(* Logix 5000 project; controller NSH_PLC1 vendor 1 type 14 code 167 rev 32.11; software revision 32.02; part 2 of 12 *)
(* tags used below, declared in another part *)
   FaultReset : BOOL;   // Huller-Sheller Fault Reset
   Num_Faults : DINT;   // Number of Huller-Sheller Faults
   Num_Warnings : DINT;   // Number of Huller-Sheller Warnings
   TempCommAlarm : BOOL;   // Temp Motor, AOP communications Alarm
   TempImbalanceTrip : BOOL;   // Temp Motor, Phase Imbalance Trip
   TempImbalanceWarning : BOOL;   // Temp Motor, Phase Imbalance Warning
   TempMotor : Motor;   // Temp Motor Tag for Subroutines
   TempOverloadTrip : BOOL;   // Temp Motor, Overload Trip
   TempOverloadWarning : BOOL;   // Temp Motor, Overlaod Warning
   TempPhaseLossTrip : BOOL;   // Temp Motor, Phase Loss Trip
   TempReady : BOOL;   // Temp Motor is ready
   TempRunning : BOOL;   // Temp Motor is Running
   TempTriped : BOOL;   // Temp Motor Tripped
   TempWarning : BOOL;   // Temp Motor Warning
   AFI : BOOL;   // Always False
   BH1 : Motor;   // Auger
   BH1D : Motor;   // Airlock
   BH2 : Motor;   // S. Ele
   BH2D : Motor;   // Airlock
   BH3D : Motor;   // Airlock
   C10 : Motor;   // Auger
   C1A : Motor;   // Auger
   C1B : Motor;   // Auger
   C2 : Motor;   // Auger
   C3A : Motor;   // Auger
   C3B : Motor;   // Auger
   C4 : Motor;   // Ele.
   C7 : Motor;   // Ele
   C8 : Motor;   // Auger
   C9 : Motor;   // Auger
   CL1 : Motor;   // Auger
   CL2 : Motor;   // Auger
   CL3 : Motor;   // Auger
   CL4 : Motor;   // Auger
   CL5 : Motor;   // Auger
   CL6 : Motor;   // Auger
   D10 : Motor;   // Ele
   D11 : Motor;   // Auger
   D12 : Motor;   // Auger
   D13 : Motor;   // Auger
   D14 : Motor;   // Auger
   D1A : Motor;   // Auger
   D1B : Motor;   // Auger
   D2 : Motor;   // Auger
   D4 : Motor;   // Auger
   D5 : Motor;   // Auger
   D6 : Motor;   // Auger
   DL1 : Motor;   // Auger
   M20 : Motor;   // Ele.
   M21 : Motor;   // Nolin
   M25 : Motor;   // Accept Vib.
   M42C : Motor;   // 3C Deck
   M42D : Motor;   // 3C Deck
   M43CA : Motor;   // Asp.
   M43CB : Motor;   // Asp.
   M43DA : Motor;   // Asp.
   M43DB : Motor;   // Asp.
   S11 : Motor;   // Ele.
   S12 : Motor;   // Auger
   S47 : Motor;   // Auger
   S48 : Motor;   // Auger
   S49 : Motor;   // Auger
   S50 : Motor;   // Auger
   SL1 : Motor;   // Auger
   T1 : Motor;   // Belt
   T2 : Motor;   // Belt
   T3 : Motor;   // Belt
   TMR_StartHS : TIMER;   // Run Hullers & Shellers Warning Timer
(* HullerSheller, continued *)

ROUTINE E300_StatusAlmWarnSUB   (* ladder *)
// Decode Status Bits and Set Warnings and Alarms For NRFV Motors with E300
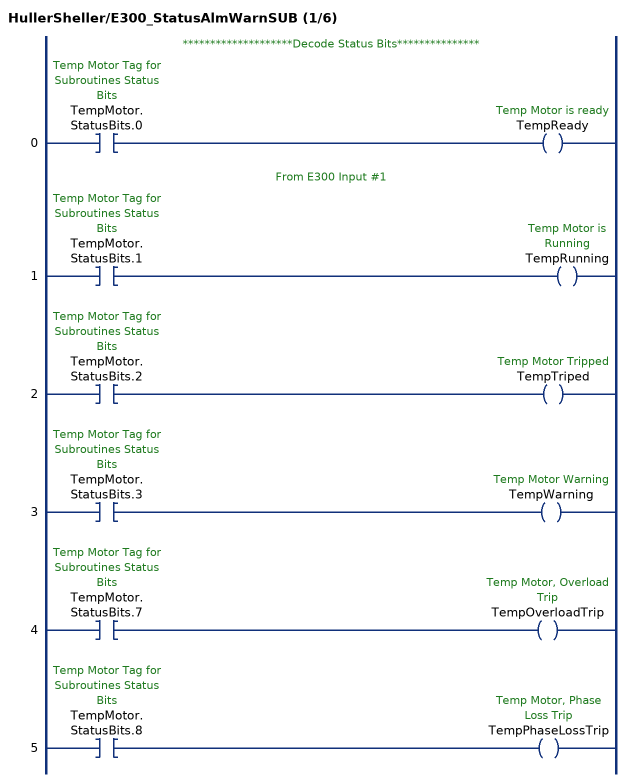
   // ********************Decode Status Bits***************
   0: XIC(TempMotor.StatusBits.0)OTE(TempReady);
   // From E300 Input #1
   1: XIC(TempMotor.StatusBits.1)OTE(TempRunning);
   2: XIC(TempMotor.StatusBits.2)OTE(TempTriped);
   3: XIC(TempMotor.StatusBits.3)OTE(TempWarning);
   4: XIC(TempMotor.StatusBits.7)OTE(TempOverloadTrip);
   5: XIC(TempMotor.StatusBits.8)OTE(TempPhaseLossTrip);
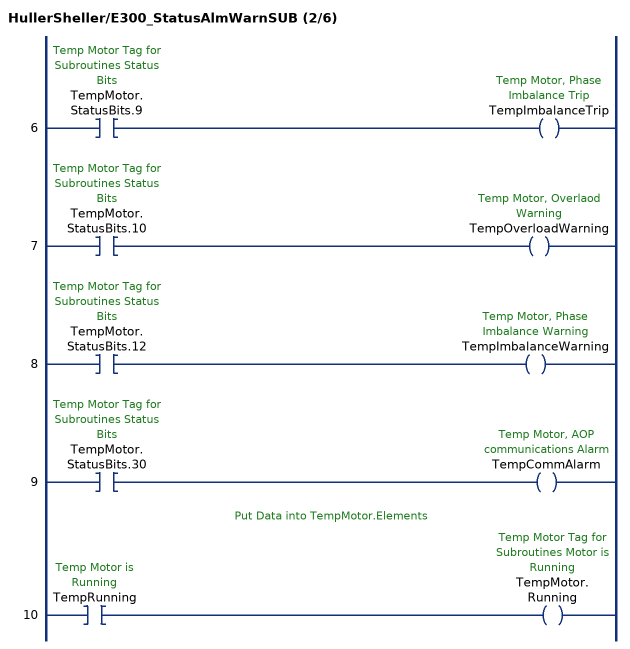
   6: XIC(TempMotor.StatusBits.9)OTE(TempImbalanceTrip);
   7: XIC(TempMotor.StatusBits.10)OTE(TempOverloadWarning);
   8: XIC(TempMotor.StatusBits.12)OTE(TempImbalanceWarning);
   9: XIC(TempMotor.StatusBits.30)OTE(TempCommAlarm);
   // Put Data into TempMotor.Elements
   10: XIC(TempRunning)OTE(TempMotor.Running);
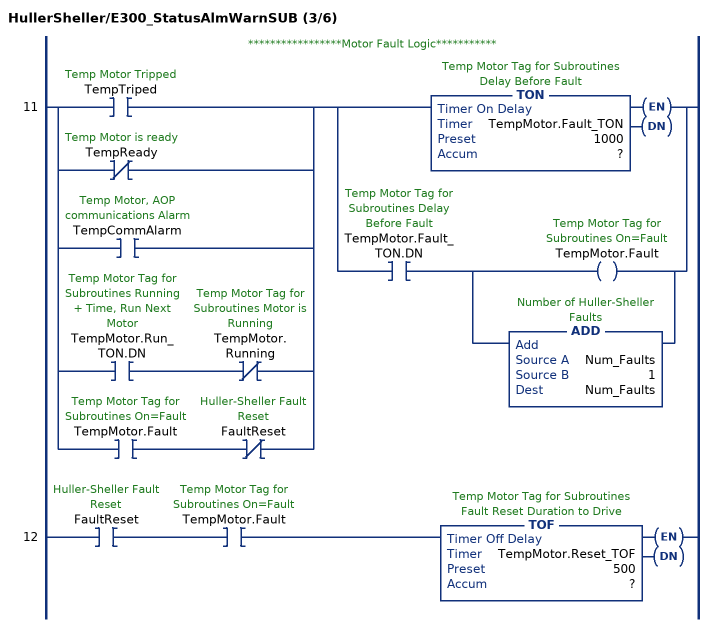
   // *****************Motor Fault Logic***********
   11: [XIC(TempTriped) ,XIO(TempReady) ,XIC(TempCommAlarm) ,XIC(TempMotor.Run_TON.DN) XIO(TempMotor.Running) ,XIC(TempMotor.Fault) XIO(FaultReset) ][TON(TempMotor.Fault_TON,?,?) ,XIC(TempMotor.Fault_TON.DN) [OTE(TempMotor.Fault) ,ADD(Num_Faults,1,Num_Faults) ] ];
   12: XIC(FaultReset)XIC(TempMotor.Fault)TOF(TempMotor.Reset_TOF,?,?);
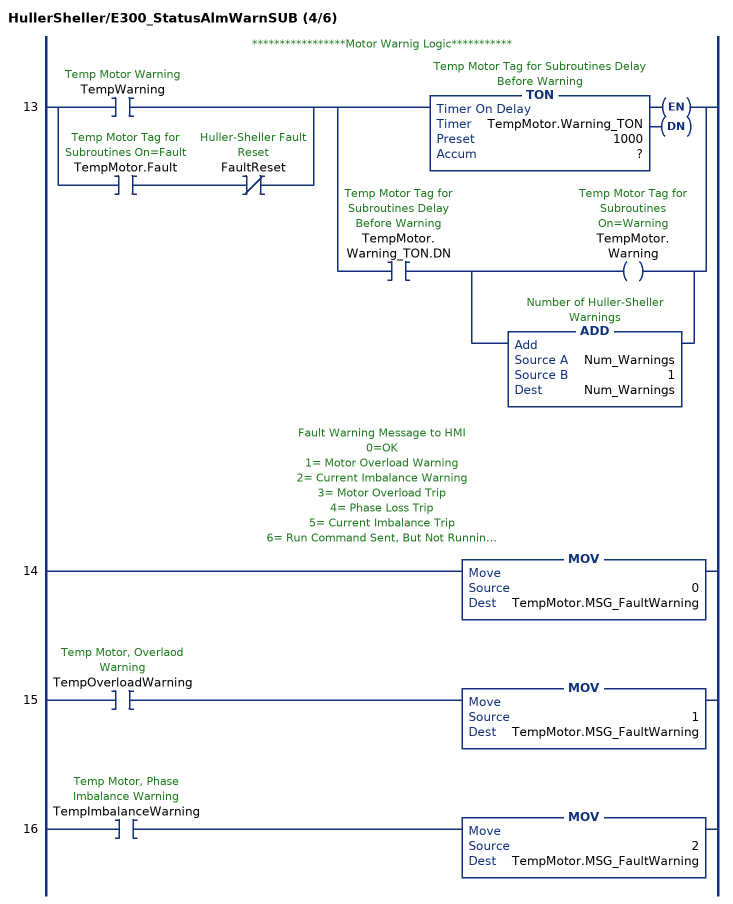
   // *****************Motor Warnig Logic***********
   13: [XIC(TempWarning) ,XIC(TempMotor.Fault) XIO(FaultReset) ][TON(TempMotor.Warning_TON,?,?) ,XIC(TempMotor.Warning_TON.DN) [OTE(TempMotor.Warning) ,ADD(Num_Warnings,1,Num_Warnings) ] ];
   // Fault Warning Message to HMI
   // 0=OK
   // 1= Motor Overload Warning
   // 2= Current Imbalance Warning
   // 3= Motor Overload Trip
   // 4= Phase Loss Trip
   // 5= Current Imbalance Trip
   // 6= Run Command Sent, But Not Running
   // 7=Loss Of Ethernet Communications
   // 8=VFD Fault
   14: MOV(0,TempMotor.MSG_FaultWarning);
   15: XIC(TempOverloadWarning)MOV(1,TempMotor.MSG_FaultWarning);
   16: XIC(TempImbalanceWarning)MOV(2,TempMotor.MSG_FaultWarning);
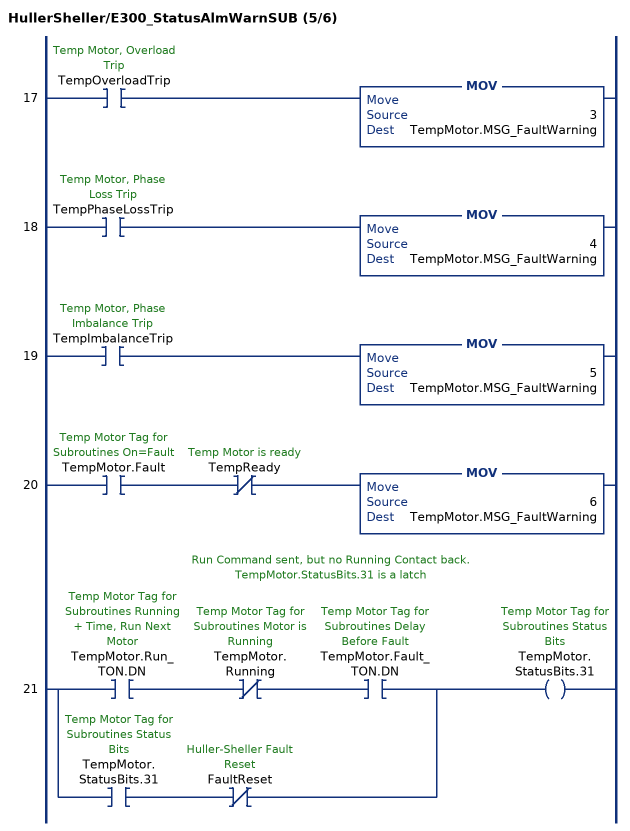
   17: XIC(TempOverloadTrip)MOV(3,TempMotor.MSG_FaultWarning);
   18: XIC(TempPhaseLossTrip)MOV(4,TempMotor.MSG_FaultWarning);
   19: XIC(TempImbalanceTrip)MOV(5,TempMotor.MSG_FaultWarning);
   20: XIC(TempMotor.Fault)XIO(TempReady)MOV(6,TempMotor.MSG_FaultWarning);
   // Run Command sent, but no Running Contact back.
   // TempMotor.StatusBits.31 is a latch
   21: [XIC(TempMotor.Run_TON.DN) XIO(TempMotor.Running) XIC(TempMotor.Fault_TON.DN) ,XIC(TempMotor.StatusBits.31) XIO(FaultReset) ]OTE(TempMotor.StatusBits.31);
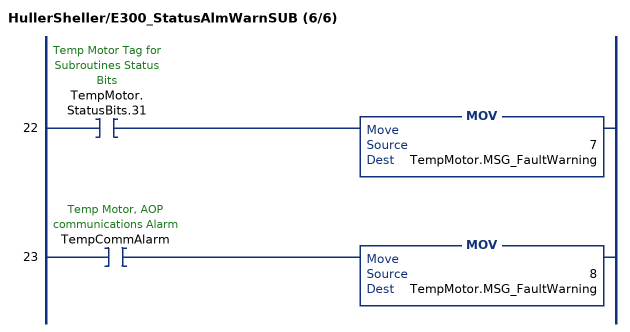
   22: XIC(TempMotor.StatusBits.31)MOV(7,TempMotor.MSG_FaultWarning);
   23: XIC(TempCommAlarm)MOV(8,TempMotor.MSG_FaultWarning);
END_ROUTINE

ROUTINE HS_MainJSR   (* ladder *)
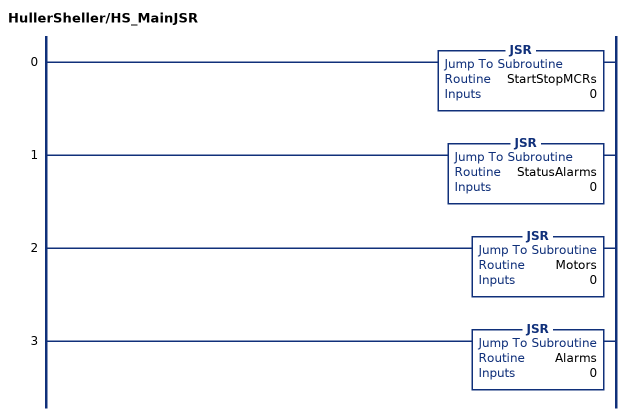
   0: JSR(StartStopMCRs,0);
   1: JSR(StatusAlarms,0);
   2: JSR(Motors,0);
   3: JSR(Alarms,0);
END_ROUTINE

ROUTINE Motors   (* ladder *)
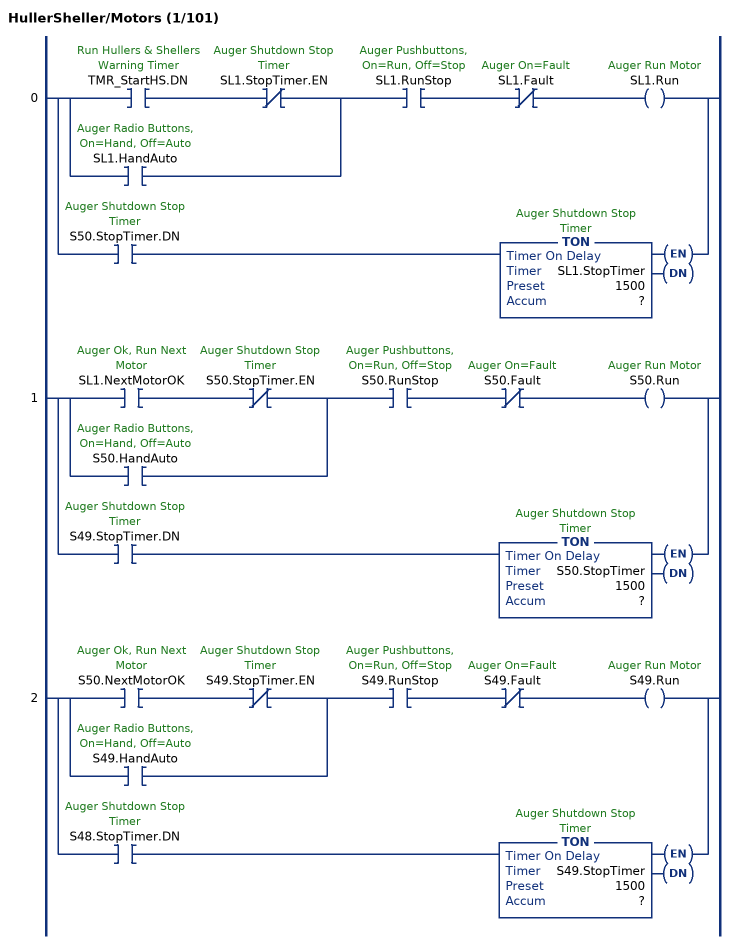
   0: [[XIC(TMR_StartHS.DN) XIO(SL1.StopTimer.EN) ,XIC(SL1.HandAuto) ] XIC(SL1.RunStop) XIO(SL1.Fault) OTE(SL1.Run) ,XIC(S50.StopTimer.DN) TON(SL1.StopTimer,?,?) ];
   1: [[XIC(SL1.NextMotorOK) XIO(S50.StopTimer.EN) ,XIC(S50.HandAuto) ] XIC(S50.RunStop) XIO(S50.Fault) OTE(S50.Run) ,XIC(S49.StopTimer.DN) TON(S50.StopTimer,?,?) ];
   2: [[XIC(S50.NextMotorOK) XIO(S49.StopTimer.EN) ,XIC(S49.HandAuto) ] XIC(S49.RunStop) XIO(S49.Fault) OTE(S49.Run) ,XIC(S48.StopTimer.DN) TON(S49.StopTimer,?,?) ];
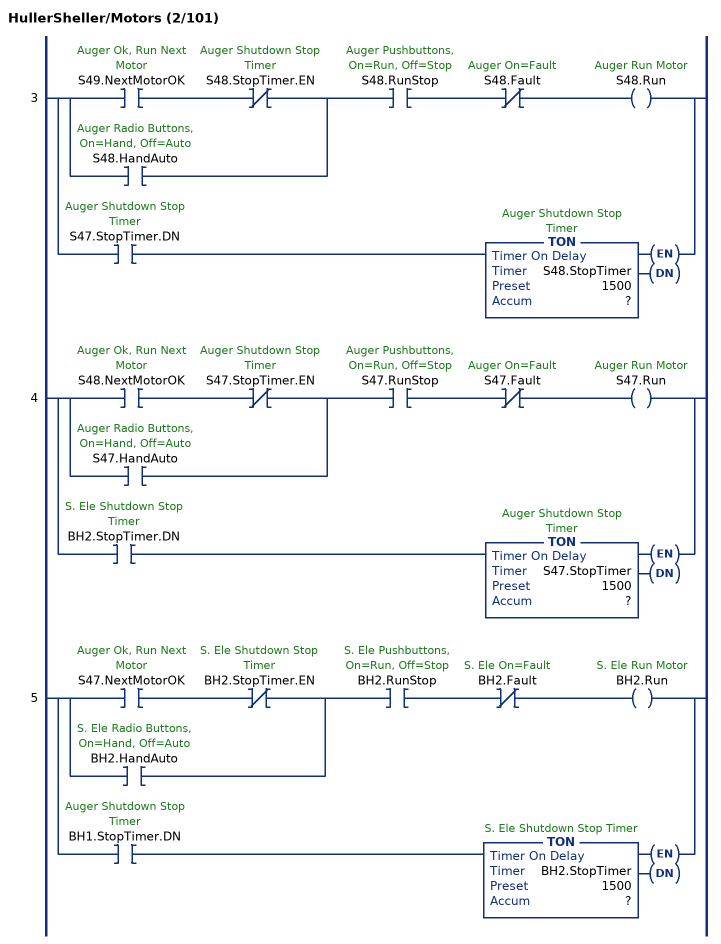
   3: [[XIC(S49.NextMotorOK) XIO(S48.StopTimer.EN) ,XIC(S48.HandAuto) ] XIC(S48.RunStop) XIO(S48.Fault) OTE(S48.Run) ,XIC(S47.StopTimer.DN) TON(S48.StopTimer,?,?) ];
   4: [[XIC(S48.NextMotorOK) XIO(S47.StopTimer.EN) ,XIC(S47.HandAuto) ] XIC(S47.RunStop) XIO(S47.Fault) OTE(S47.Run) ,XIC(BH2.StopTimer.DN) TON(S47.StopTimer,?,?) ];
   5: [[XIC(S47.NextMotorOK) XIO(BH2.StopTimer.EN) ,XIC(BH2.HandAuto) ] XIC(BH2.RunStop) XIO(BH2.Fault) OTE(BH2.Run) ,XIC(BH1.StopTimer.DN) TON(BH2.StopTimer,?,?) ];
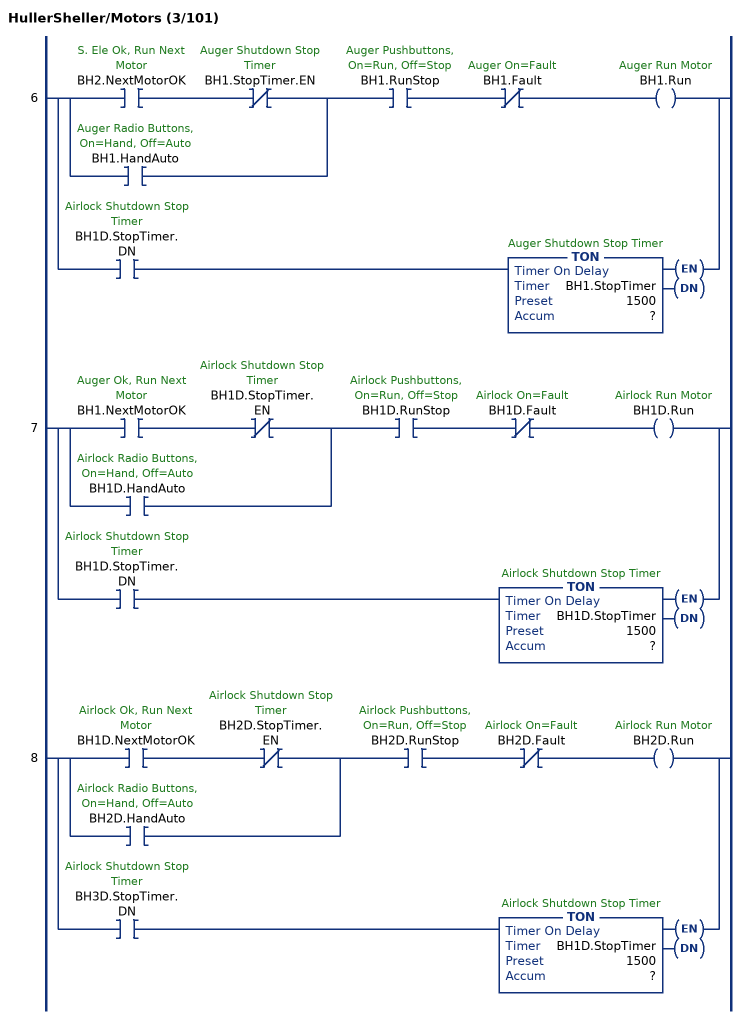
   6: [[XIC(BH2.NextMotorOK) XIO(BH1.StopTimer.EN) ,XIC(BH1.HandAuto) ] XIC(BH1.RunStop) XIO(BH1.Fault) OTE(BH1.Run) ,XIC(BH1D.StopTimer.DN) TON(BH1.StopTimer,?,?) ];
   7: [[XIC(BH1.NextMotorOK) XIO(BH1D.StopTimer.EN) ,XIC(BH1D.HandAuto) ] XIC(BH1D.RunStop) XIO(BH1D.Fault) OTE(BH1D.Run) ,XIC(BH1D.StopTimer.DN) TON(BH1D.StopTimer,?,?) ];
   8: [[XIC(BH1D.NextMotorOK) XIO(BH2D.StopTimer.EN) ,XIC(BH2D.HandAuto) ] XIC(BH2D.RunStop) XIO(BH2D.Fault) OTE(BH2D.Run) ,XIC(BH3D.StopTimer.DN) TON(BH1D.StopTimer,?,?) ];
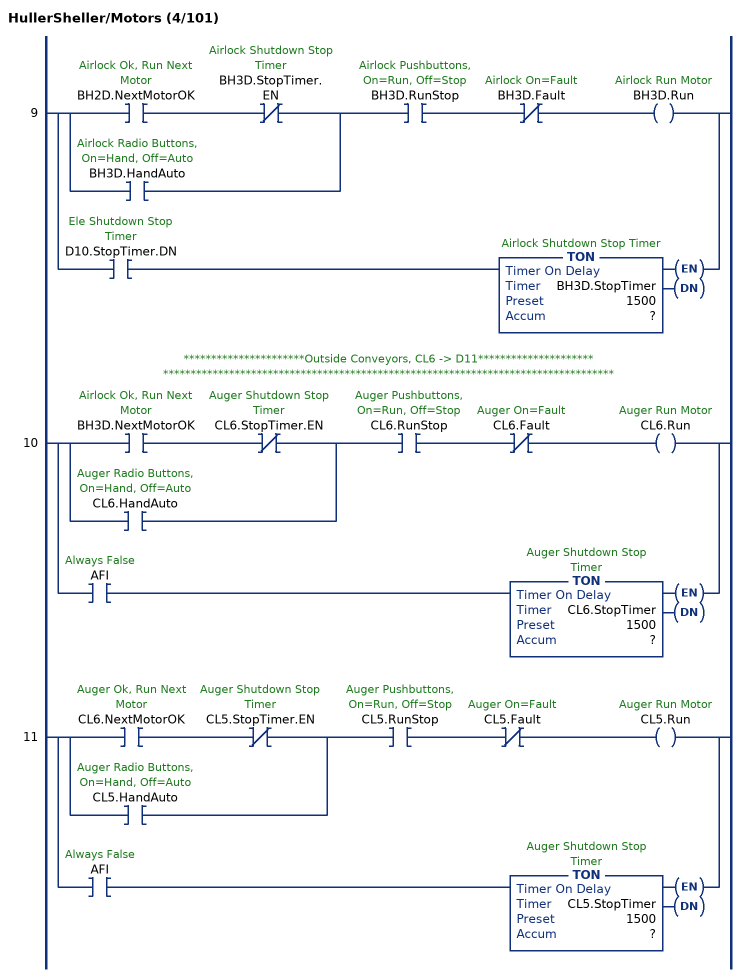
   9: [[XIC(BH2D.NextMotorOK) XIO(BH3D.StopTimer.EN) ,XIC(BH3D.HandAuto) ] XIC(BH3D.RunStop) XIO(BH3D.Fault) OTE(BH3D.Run) ,XIC(D10.StopTimer.DN) TON(BH3D.StopTimer,?,?) ];
   // **********************Outside Conveyors, CL6 -> D11*********************
   // **********************************************************************************
   10: [[XIC(BH3D.NextMotorOK) XIO(CL6.StopTimer.EN) ,XIC(CL6.HandAuto) ] XIC(CL6.RunStop) XIO(CL6.Fault) OTE(CL6.Run) ,XIC(AFI) TON(CL6.StopTimer,?,?) ];
   11: [[XIC(CL6.NextMotorOK) XIO(CL5.StopTimer.EN) ,XIC(CL5.HandAuto) ] XIC(CL5.RunStop) XIO(CL5.Fault) OTE(CL5.Run) ,XIC(AFI) TON(CL5.StopTimer,?,?) ];
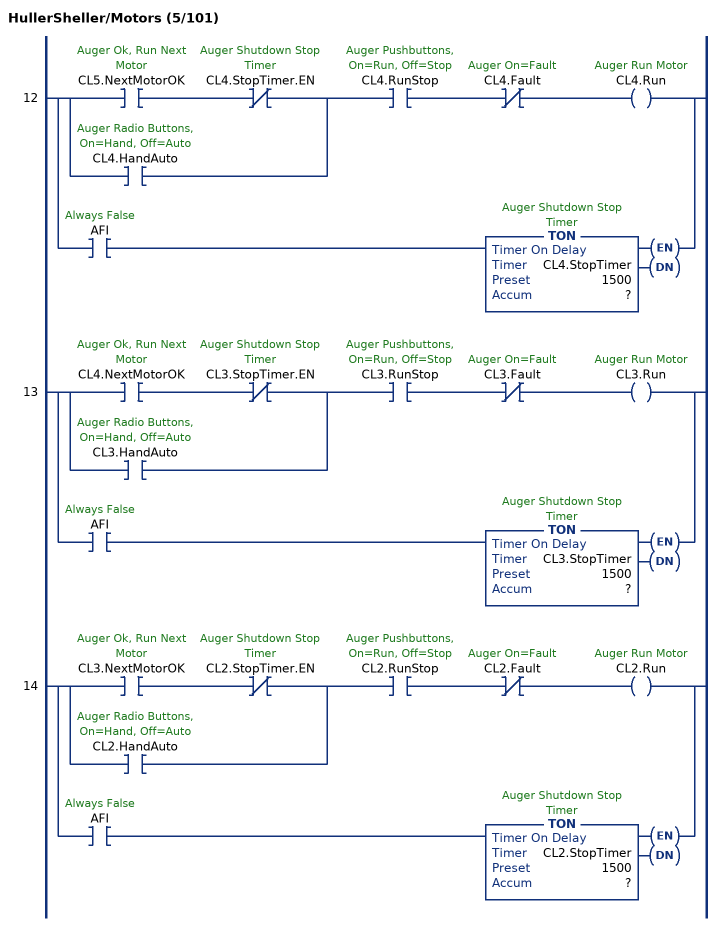
   12: [[XIC(CL5.NextMotorOK) XIO(CL4.StopTimer.EN) ,XIC(CL4.HandAuto) ] XIC(CL4.RunStop) XIO(CL4.Fault) OTE(CL4.Run) ,XIC(AFI) TON(CL4.StopTimer,?,?) ];
   13: [[XIC(CL4.NextMotorOK) XIO(CL3.StopTimer.EN) ,XIC(CL3.HandAuto) ] XIC(CL3.RunStop) XIO(CL3.Fault) OTE(CL3.Run) ,XIC(AFI) TON(CL3.StopTimer,?,?) ];
   14: [[XIC(CL3.NextMotorOK) XIO(CL2.StopTimer.EN) ,XIC(CL2.HandAuto) ] XIC(CL2.RunStop) XIO(CL2.Fault) OTE(CL2.Run) ,XIC(AFI) TON(CL2.StopTimer,?,?) ];
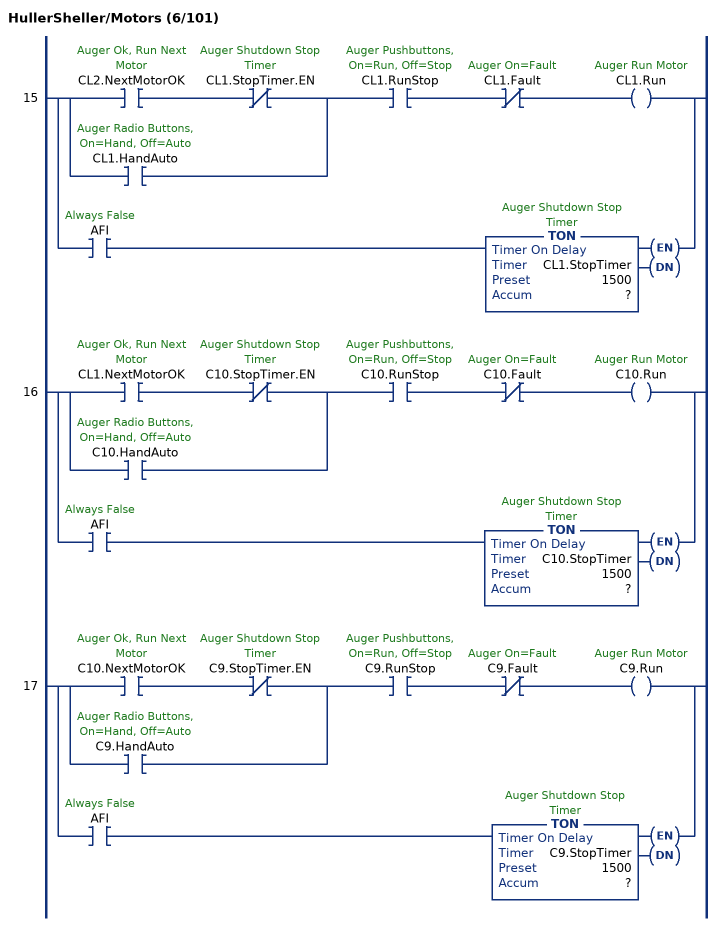
   15: [[XIC(CL2.NextMotorOK) XIO(CL1.StopTimer.EN) ,XIC(CL1.HandAuto) ] XIC(CL1.RunStop) XIO(CL1.Fault) OTE(CL1.Run) ,XIC(AFI) TON(CL1.StopTimer,?,?) ];
   16: [[XIC(CL1.NextMotorOK) XIO(C10.StopTimer.EN) ,XIC(C10.HandAuto) ] XIC(C10.RunStop) XIO(C10.Fault) OTE(C10.Run) ,XIC(AFI) TON(C10.StopTimer,?,?) ];
   17: [[XIC(C10.NextMotorOK) XIO(C9.StopTimer.EN) ,XIC(C9.HandAuto) ] XIC(C9.RunStop) XIO(C9.Fault) OTE(C9.Run) ,XIC(AFI) TON(C9.StopTimer,?,?) ];
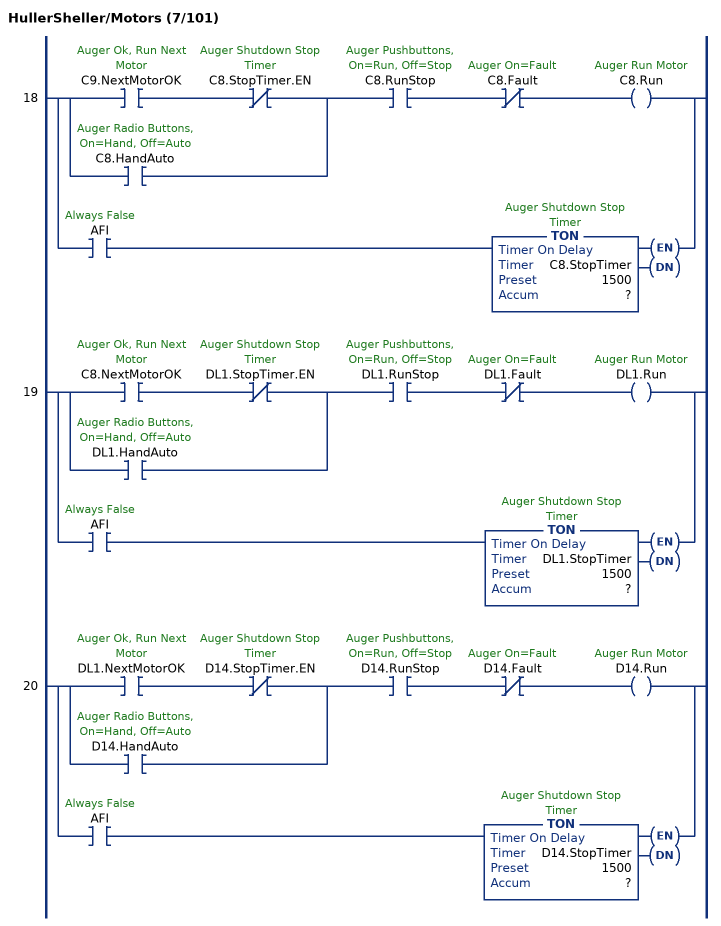
   18: [[XIC(C9.NextMotorOK) XIO(C8.StopTimer.EN) ,XIC(C8.HandAuto) ] XIC(C8.RunStop) XIO(C8.Fault) OTE(C8.Run) ,XIC(AFI) TON(C8.StopTimer,?,?) ];
   19: [[XIC(C8.NextMotorOK) XIO(DL1.StopTimer.EN) ,XIC(DL1.HandAuto) ] XIC(DL1.RunStop) XIO(DL1.Fault) OTE(DL1.Run) ,XIC(AFI) TON(DL1.StopTimer,?,?) ];
   20: [[XIC(DL1.NextMotorOK) XIO(D14.StopTimer.EN) ,XIC(D14.HandAuto) ] XIC(D14.RunStop) XIO(D14.Fault) OTE(D14.Run) ,XIC(AFI) TON(D14.StopTimer,?,?) ];
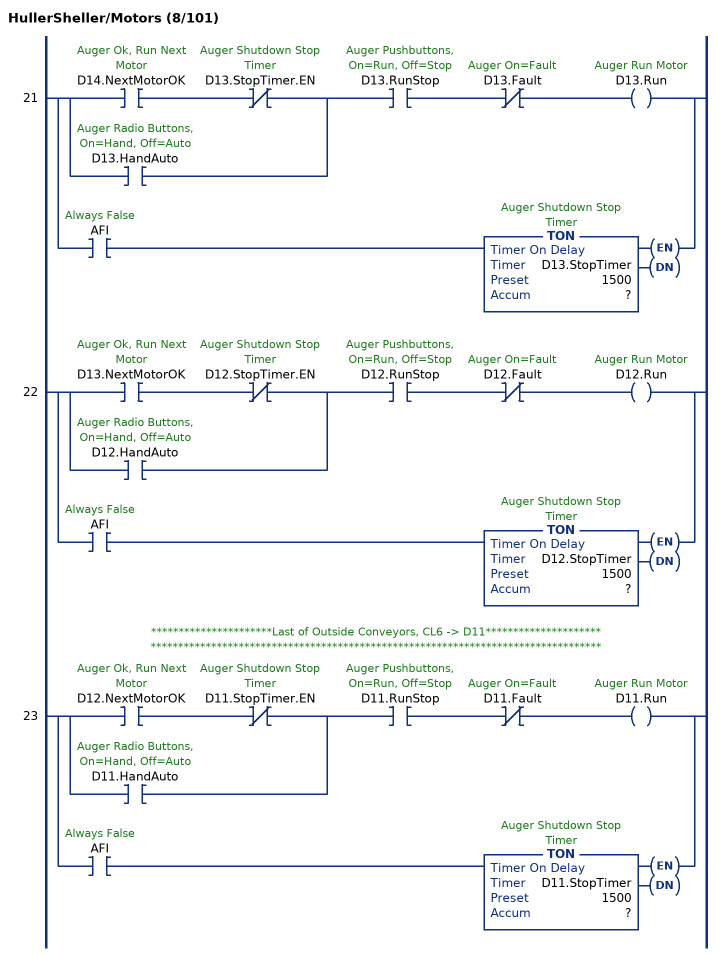
   21: [[XIC(D14.NextMotorOK) XIO(D13.StopTimer.EN) ,XIC(D13.HandAuto) ] XIC(D13.RunStop) XIO(D13.Fault) OTE(D13.Run) ,XIC(AFI) TON(D13.StopTimer,?,?) ];
   22: [[XIC(D13.NextMotorOK) XIO(D12.StopTimer.EN) ,XIC(D12.HandAuto) ] XIC(D12.RunStop) XIO(D12.Fault) OTE(D12.Run) ,XIC(AFI) TON(D12.StopTimer,?,?) ];
   // **********************Last of Outside Conveyors, CL6 -> D11*********************
   // **********************************************************************************
   23: [[XIC(D12.NextMotorOK) XIO(D11.StopTimer.EN) ,XIC(D11.HandAuto) ] XIC(D11.RunStop) XIO(D11.Fault) OTE(D11.Run) ,XIC(AFI) TON(D11.StopTimer,?,?) ];
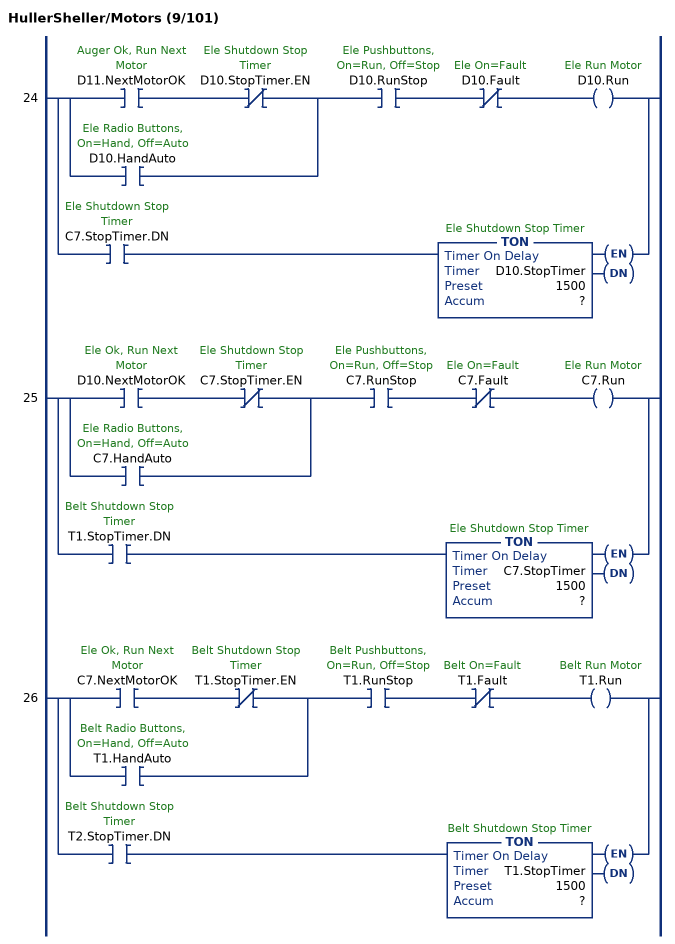
   24: [[XIC(D11.NextMotorOK) XIO(D10.StopTimer.EN) ,XIC(D10.HandAuto) ] XIC(D10.RunStop) XIO(D10.Fault) OTE(D10.Run) ,XIC(C7.StopTimer.DN) TON(D10.StopTimer,?,?) ];
   25: [[XIC(D10.NextMotorOK) XIO(C7.StopTimer.EN) ,XIC(C7.HandAuto) ] XIC(C7.RunStop) XIO(C7.Fault) OTE(C7.Run) ,XIC(T1.StopTimer.DN) TON(C7.StopTimer,?,?) ];
   26: [[XIC(C7.NextMotorOK) XIO(T1.StopTimer.EN) ,XIC(T1.HandAuto) ] XIC(T1.RunStop) XIO(T1.Fault) OTE(T1.Run) ,XIC(T2.StopTimer.DN) TON(T1.StopTimer,?,?) ];
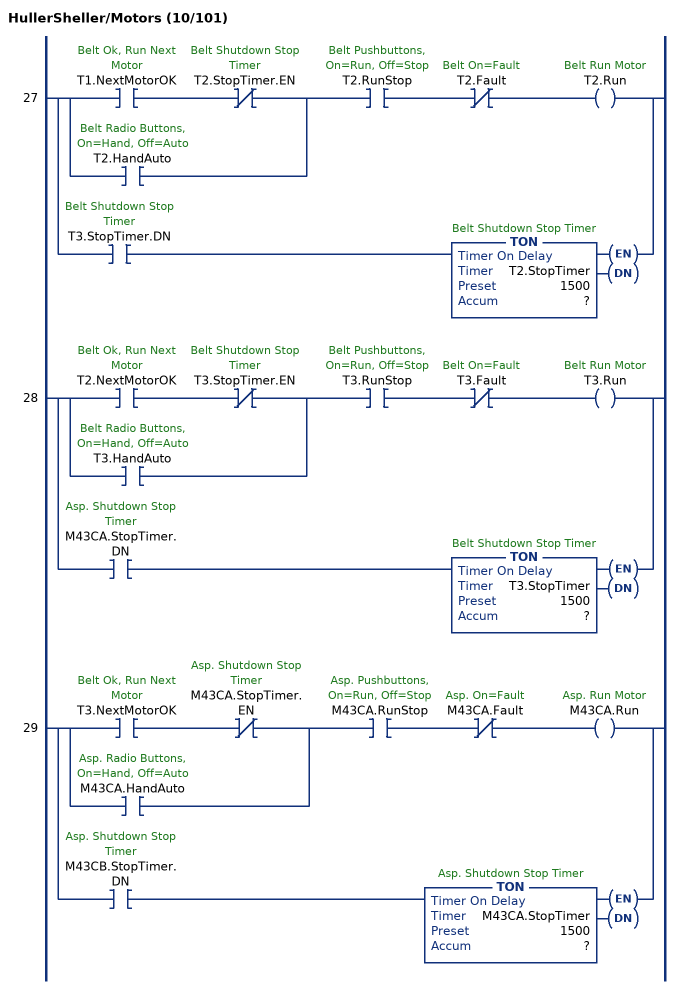
   27: [[XIC(T1.NextMotorOK) XIO(T2.StopTimer.EN) ,XIC(T2.HandAuto) ] XIC(T2.RunStop) XIO(T2.Fault) OTE(T2.Run) ,XIC(T3.StopTimer.DN) TON(T2.StopTimer,?,?) ];
   28: [[XIC(T2.NextMotorOK) XIO(T3.StopTimer.EN) ,XIC(T3.HandAuto) ] XIC(T3.RunStop) XIO(T3.Fault) OTE(T3.Run) ,XIC(M43CA.StopTimer.DN) TON(T3.StopTimer,?,?) ];
   29: [[XIC(T3.NextMotorOK) XIO(M43CA.StopTimer.EN) ,XIC(M43CA.HandAuto) ] XIC(M43CA.RunStop) XIO(M43CA.Fault) OTE(M43CA.Run) ,XIC(M43CB.StopTimer.DN) TON(M43CA.StopTimer,?,?) ];
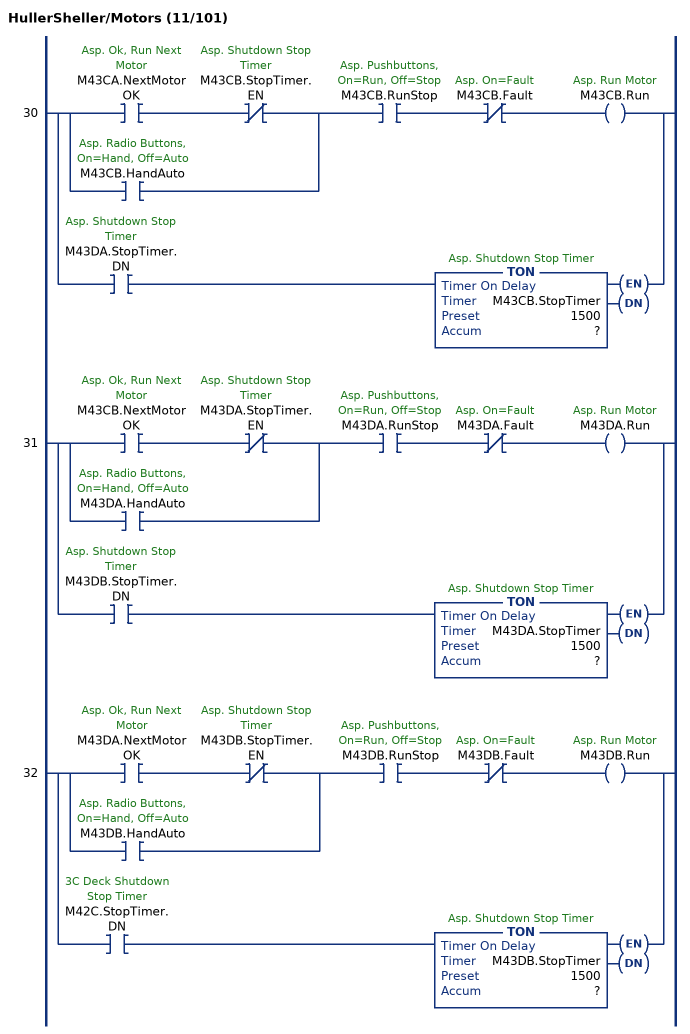
   30: [[XIC(M43CA.NextMotorOK) XIO(M43CB.StopTimer.EN) ,XIC(M43CB.HandAuto) ] XIC(M43CB.RunStop) XIO(M43CB.Fault) OTE(M43CB.Run) ,XIC(M43DA.StopTimer.DN) TON(M43CB.StopTimer,?,?) ];
   31: [[XIC(M43CB.NextMotorOK) XIO(M43DA.StopTimer.EN) ,XIC(M43DA.HandAuto) ] XIC(M43DA.RunStop) XIO(M43DA.Fault) OTE(M43DA.Run) ,XIC(M43DB.StopTimer.DN) TON(M43DA.StopTimer,?,?) ];
   32: [[XIC(M43DA.NextMotorOK) XIO(M43DB.StopTimer.EN) ,XIC(M43DB.HandAuto) ] XIC(M43DB.RunStop) XIO(M43DB.Fault) OTE(M43DB.Run) ,XIC(M42C.StopTimer.DN) TON(M43DB.StopTimer,?,?) ];
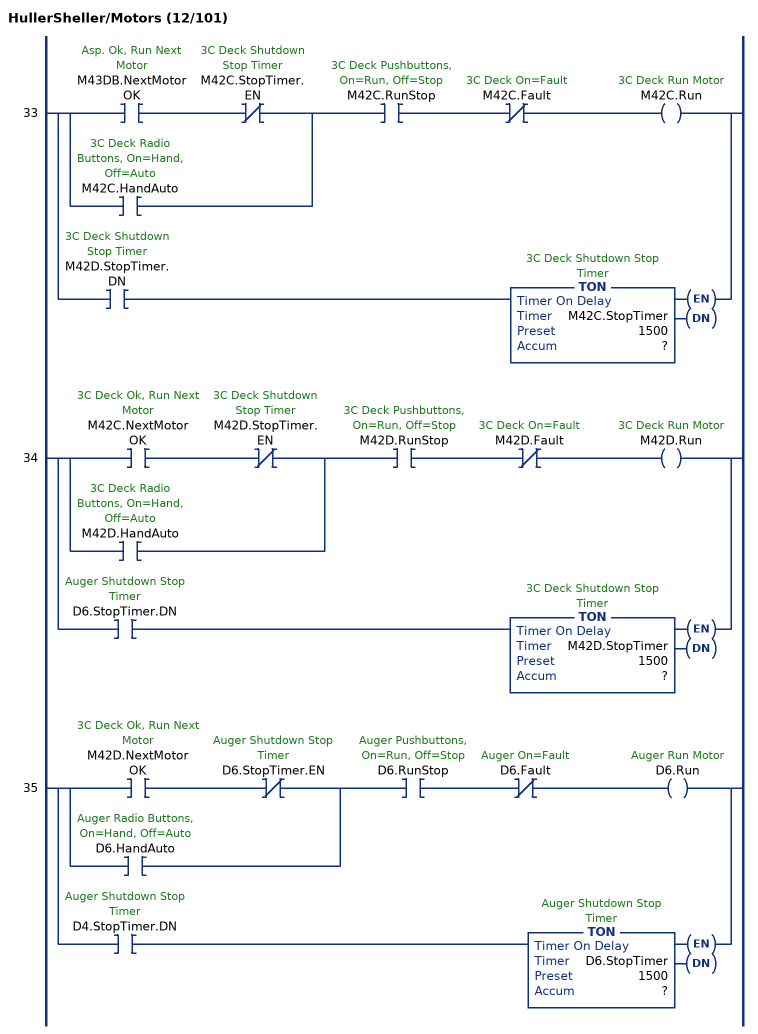
   33: [[XIC(M43DB.NextMotorOK) XIO(M42C.StopTimer.EN) ,XIC(M42C.HandAuto) ] XIC(M42C.RunStop) XIO(M42C.Fault) OTE(M42C.Run) ,XIC(M42D.StopTimer.DN) TON(M42C.StopTimer,?,?) ];
   34: [[XIC(M42C.NextMotorOK) XIO(M42D.StopTimer.EN) ,XIC(M42D.HandAuto) ] XIC(M42D.RunStop) XIO(M42D.Fault) OTE(M42D.Run) ,XIC(D6.StopTimer.DN) TON(M42D.StopTimer,?,?) ];
   35: [[XIC(M42D.NextMotorOK) XIO(D6.StopTimer.EN) ,XIC(D6.HandAuto) ] XIC(D6.RunStop) XIO(D6.Fault) OTE(D6.Run) ,XIC(D4.StopTimer.DN) TON(D6.StopTimer,?,?) ];
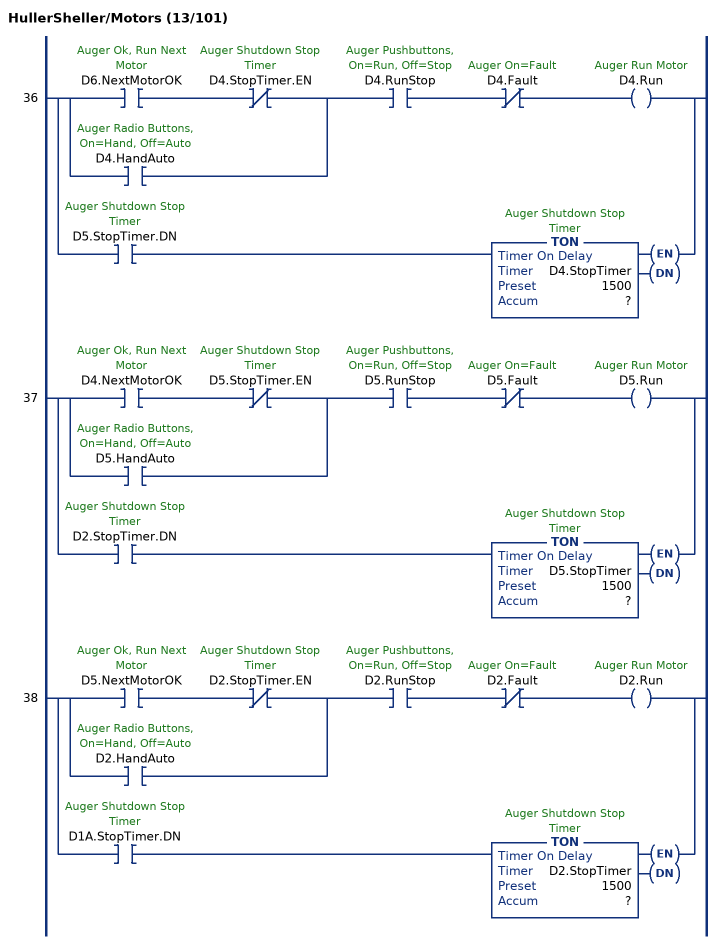
   36: [[XIC(D6.NextMotorOK) XIO(D4.StopTimer.EN) ,XIC(D4.HandAuto) ] XIC(D4.RunStop) XIO(D4.Fault) OTE(D4.Run) ,XIC(D5.StopTimer.DN) TON(D4.StopTimer,?,?) ];
   37: [[XIC(D4.NextMotorOK) XIO(D5.StopTimer.EN) ,XIC(D5.HandAuto) ] XIC(D5.RunStop) XIO(D5.Fault) OTE(D5.Run) ,XIC(D2.StopTimer.DN) TON(D5.StopTimer,?,?) ];
   38: [[XIC(D5.NextMotorOK) XIO(D2.StopTimer.EN) ,XIC(D2.HandAuto) ] XIC(D2.RunStop) XIO(D2.Fault) OTE(D2.Run) ,XIC(D1A.StopTimer.DN) TON(D2.StopTimer,?,?) ];
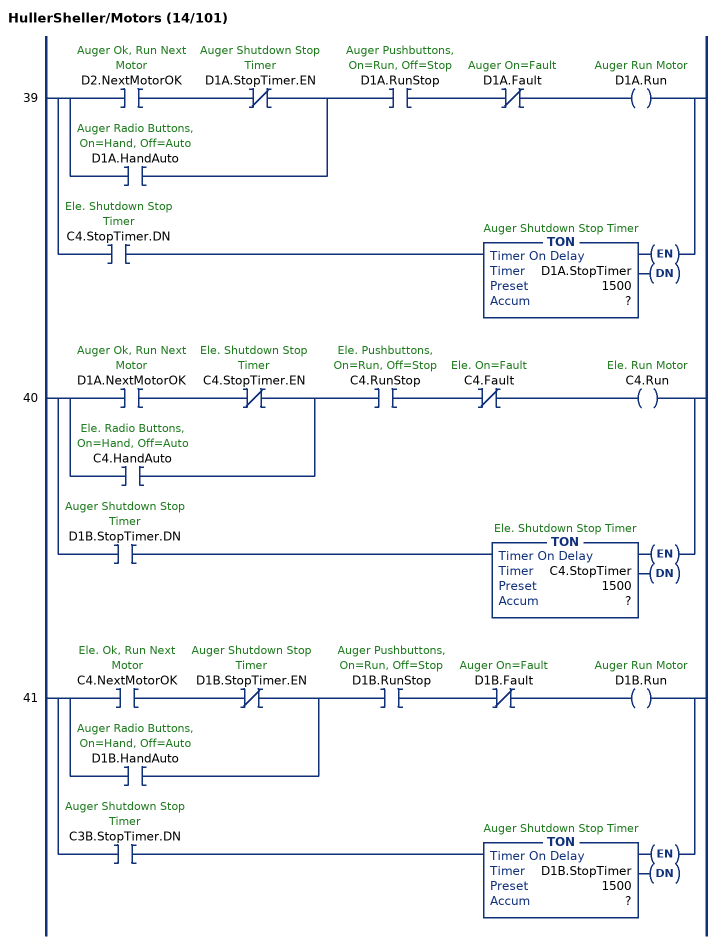
   39: [[XIC(D2.NextMotorOK) XIO(D1A.StopTimer.EN) ,XIC(D1A.HandAuto) ] XIC(D1A.RunStop) XIO(D1A.Fault) OTE(D1A.Run) ,XIC(C4.StopTimer.DN) TON(D1A.StopTimer,?,?) ];
   40: [[XIC(D1A.NextMotorOK) XIO(C4.StopTimer.EN) ,XIC(C4.HandAuto) ] XIC(C4.RunStop) XIO(C4.Fault) OTE(C4.Run) ,XIC(D1B.StopTimer.DN) TON(C4.StopTimer,?,?) ];
   41: [[XIC(C4.NextMotorOK) XIO(D1B.StopTimer.EN) ,XIC(D1B.HandAuto) ] XIC(D1B.RunStop) XIO(D1B.Fault) OTE(D1B.Run) ,XIC(C3B.StopTimer.DN) TON(D1B.StopTimer,?,?) ];
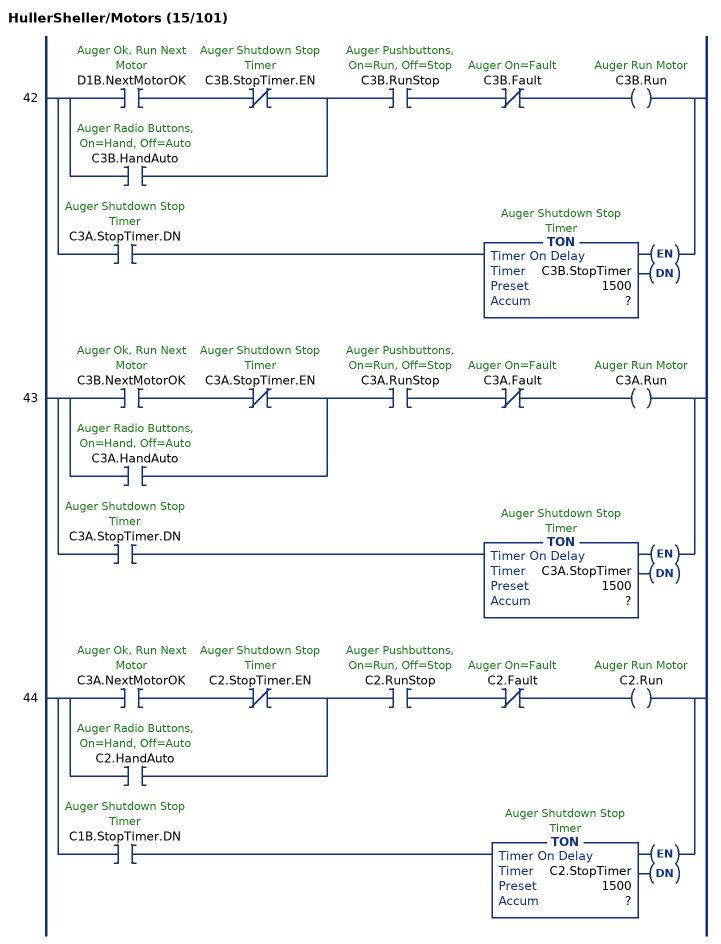
   42: [[XIC(D1B.NextMotorOK) XIO(C3B.StopTimer.EN) ,XIC(C3B.HandAuto) ] XIC(C3B.RunStop) XIO(C3B.Fault) OTE(C3B.Run) ,XIC(C3A.StopTimer.DN) TON(C3B.StopTimer,?,?) ];
   43: [[XIC(C3B.NextMotorOK) XIO(C3A.StopTimer.EN) ,XIC(C3A.HandAuto) ] XIC(C3A.RunStop) XIO(C3A.Fault) OTE(C3A.Run) ,XIC(C3A.StopTimer.DN) TON(C3A.StopTimer,?,?) ];
   44: [[XIC(C3A.NextMotorOK) XIO(C2.StopTimer.EN) ,XIC(C2.HandAuto) ] XIC(C2.RunStop) XIO(C2.Fault) OTE(C2.Run) ,XIC(C1B.StopTimer.DN) TON(C2.StopTimer,?,?) ];
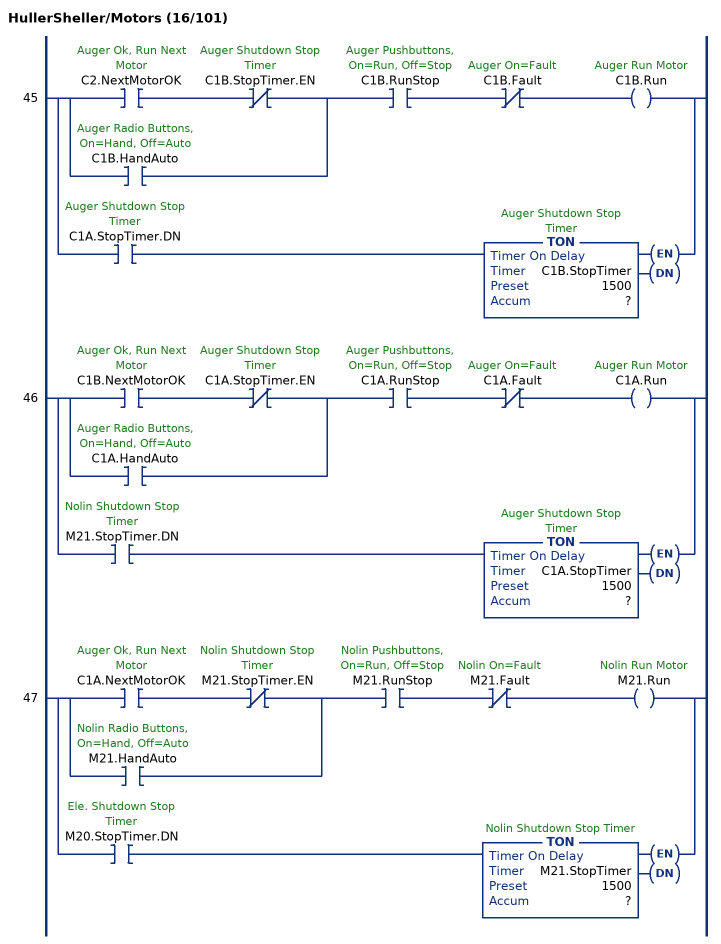
   45: [[XIC(C2.NextMotorOK) XIO(C1B.StopTimer.EN) ,XIC(C1B.HandAuto) ] XIC(C1B.RunStop) XIO(C1B.Fault) OTE(C1B.Run) ,XIC(C1A.StopTimer.DN) TON(C1B.StopTimer,?,?) ];
   46: [[XIC(C1B.NextMotorOK) XIO(C1A.StopTimer.EN) ,XIC(C1A.HandAuto) ] XIC(C1A.RunStop) XIO(C1A.Fault) OTE(C1A.Run) ,XIC(M21.StopTimer.DN) TON(C1A.StopTimer,?,?) ];
   47: [[XIC(C1A.NextMotorOK) XIO(M21.StopTimer.EN) ,XIC(M21.HandAuto) ] XIC(M21.RunStop) XIO(M21.Fault) OTE(M21.Run) ,XIC(M20.StopTimer.DN) TON(M21.StopTimer,?,?) ];
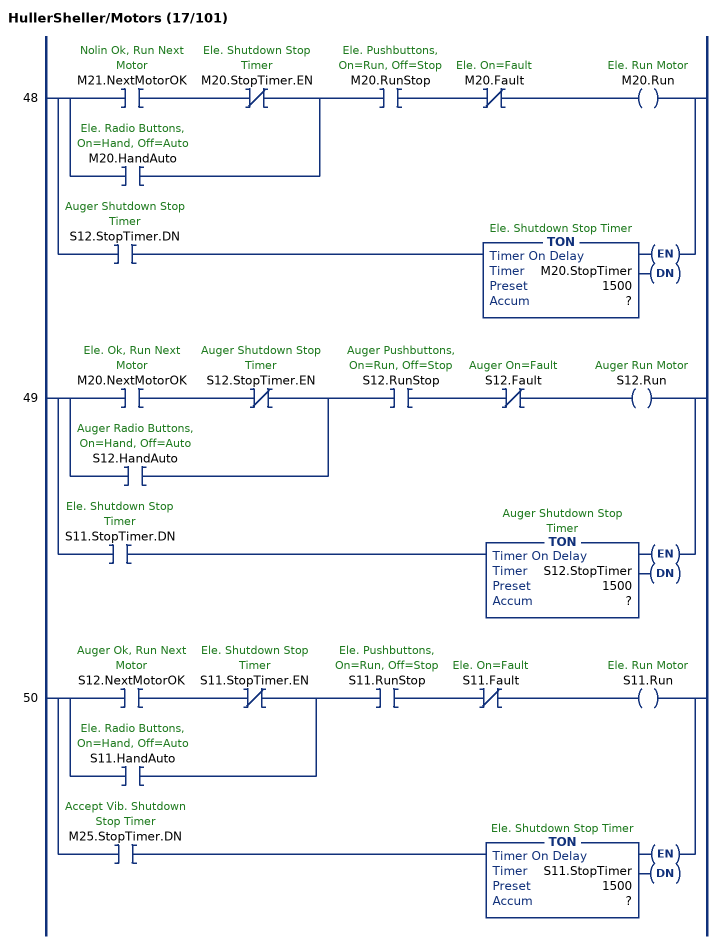
   48: [[XIC(M21.NextMotorOK) XIO(M20.StopTimer.EN) ,XIC(M20.HandAuto) ] XIC(M20.RunStop) XIO(M20.Fault) OTE(M20.Run) ,XIC(S12.StopTimer.DN) TON(M20.StopTimer,?,?) ];
   49: [[XIC(M20.NextMotorOK) XIO(S12.StopTimer.EN) ,XIC(S12.HandAuto) ] XIC(S12.RunStop) XIO(S12.Fault) OTE(S12.Run) ,XIC(S11.StopTimer.DN) TON(S12.StopTimer,?,?) ];
   50: [[XIC(S12.NextMotorOK) XIO(S11.StopTimer.EN) ,XIC(S11.HandAuto) ] XIC(S11.RunStop) XIO(S11.Fault) OTE(S11.Run) ,XIC(M25.StopTimer.DN) TON(S11.StopTimer,?,?) ];
